TYPE stSkillArray :
STRUCT
	Skills: ARRAY[1..4] OF POINTER TO FB_Skill;
END_STRUCT
END_TYPE

(* stored: Version 1.1.0.1, ProductVersion 3.1.4026.18
   DUT stSkillArray: Id {e0542c25-710d-4bb5-a626-41c90624e86c} *)
